// TIA Portal V20 export
VAR_GLOBAL   // PLC tag table "Machine"
END_VAR
VAR_GLOBAL CONSTANT   // user constants
   MC_openVice : Int := 10;
   MC_closeVice : Int := 11;
   MC_unlockPallet : Int := 20;
   MC_lockPallet : Int := 21;
   MC_openDoor : Int := 30;
   MC_closeDoor : Int := 31;
   MC_startWork : Int := 50;
   MC_unlockPartOnTable : Int := 100;
   MC_lockPartOnTable : Int := 101;
   MC_resetError : Int := 999;
END_VAR
